Staubli VAL3: Axis1Offset.pgx

public program Axis1Offset(pointRx& x_pP[], num x_nOffset, tool x_tTool)
  local num l_nNum
  local bool l_bMC
  local num l_nValue[3]
  local joint l_jJ
  local point l_pPoint
  local frame l_fFrame
begin
  if size(x_pP)<3
    return
  endIf

  for l_nNum=10 to size(x_pP)-3
    l_nValue[0]=(x_pP[l_nNum].trsf.x-x_pP[l_nNum+1].trsf.x)/(x_pP[l_nNum].trsf.x-x_pP[l_nNum+2].trsf.x)
    l_nValue[1]=(x_pP[l_nNum].trsf.y-x_pP[l_nNum+1].trsf.y)/(x_pP[l_nNum].trsf.y-x_pP[l_nNum+2].trsf.y)
    l_nValue[2]=(x_pP[l_nNum].trsf.z-x_pP[l_nNum+1].trsf.z)/(x_pP[l_nNum].trsf.z-x_pP[l_nNum+2].trsf.z)

    if l_nValue[0]!=l_nValue[1] or l_nValue[0]!=l_nValue[2]

      if !pointToJoint(x_tTool,herej(),x_pP[l_nNum],l_jJ)
        popUpMsg("转换出错")
        disablePower()
        return
      else
        l_jJ.j1=l_jJ.j1+x_nOffset
        link(l_fFrame,world)
        link(l_pPoint,world)
        l_pPoint.trsf=position(x_pP[l_nNum],world)

        l_fFrame.trsf=l_pPoint.trsf*!x_pP[l_nNum].trsf
        l_pPoint=jointToPoint(x_tTool,l_fFrame,l_jJ)
        x_pP[l_nNum].trsf=l_pPoint.trsf
      endIf




    endIf




  endFor

















end
